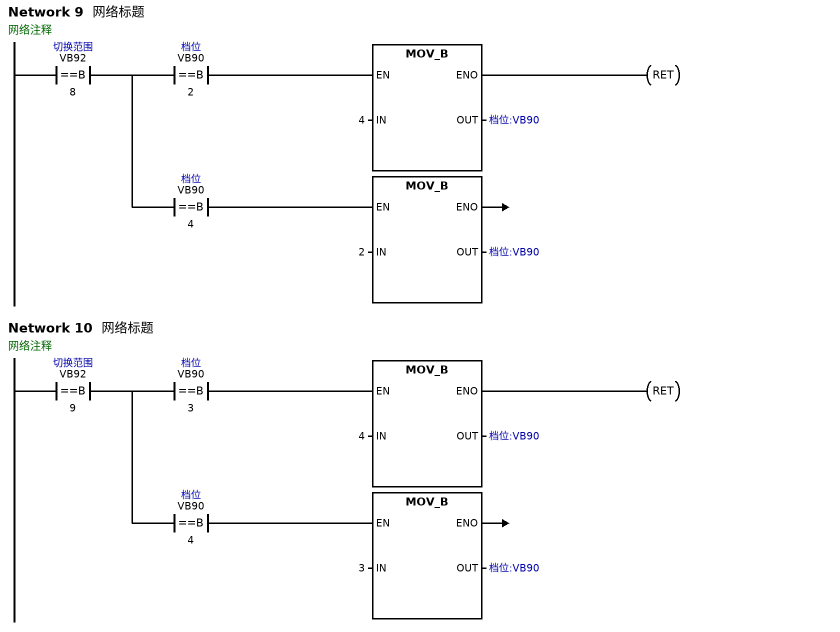
[picture p72: SBR19 networks 9-10]
Network 9 // 网络标题
// 网络注释
LDB=   切换范围:VB92, 8
LPS
AB=    档位:VB90, 2
MOVB   4, 档位:VB90
AENO
CRET
LPP
AB=    档位:VB90, 4
MOVB   2, 档位:VB90
Network 10 // 网络标题
// 网络注释
LDB=   切换范围:VB92, 9
LPS
AB=    档位:VB90, 3
MOVB   4, 档位:VB90
AENO
CRET
LPP
AB=    档位:VB90, 4
MOVB   3, 档位:VB90
END_SUBROUTINE_BLOCK

// SBR21: protected block, not included

SUBROUTINE_BLOCK ReCal:SBR22
TITLE=子程序注释
VAR_INPUT
Uo:REAL;	// LD0 
C‘:REAL;	// LD4 
K:REAL;	// LD8 
b:REAL;	// LD12 
END_VAR
VAR_OUTPUT
U‘:REAL;	// LD16 
A’:REAL;	// LD20 
END_VAR
VAR
mid:REAL;	// LD24 
END_VAR
BEGIN
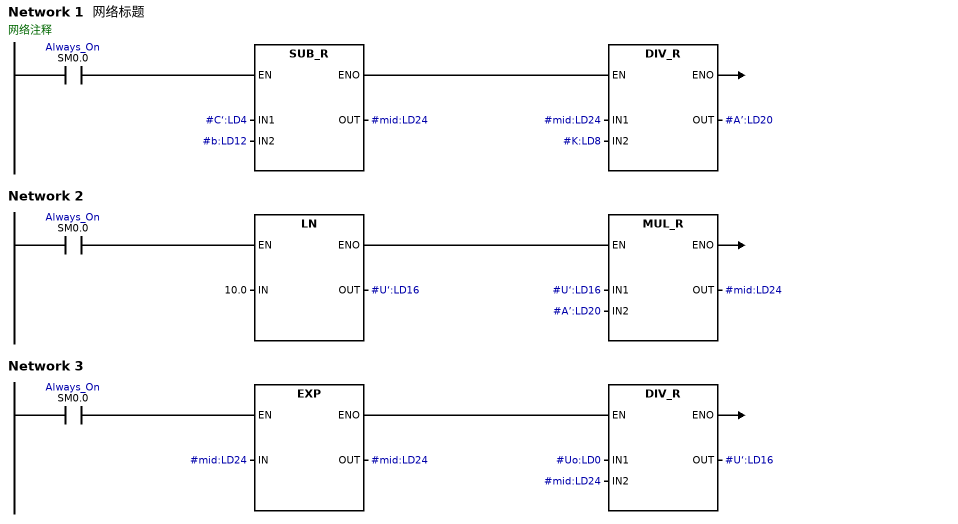
Network 1 // 网络标题
// 网络注释
LD     Always_On:SM0.0
MOVR   #C‘:LD4, #mid:LD24
AENO
-R     #b:LD12, #mid:LD24
AENO
MOVR   #mid:LD24, #A’:LD20
/R     #K:LD8, #A’:LD20
Network 2
LD     Always_On:SM0.0
LN     10.0, #U‘:LD16
AENO
MOVR   #U‘:LD16, #mid:LD24
*R     #A’:LD20, #mid:LD24
Network 3
LD     Always_On:SM0.0
EXP    #mid:LD24, #mid:LD24
AENO
MOVR   #Uo:LD0, #U‘:LD16
/R     #mid:LD24, #U‘:LD16
Network 4 // 网络标题
// 网络注释
END_SUBROUTINE_BLOCK

SUBROUTINE_BLOCK 标准R_I:SBR23
TITLE=子程序注释
VAR_INPUT
R_H:REAL;	// LD0 
R_L:REAL;	// LD4 
I_H:WORD;	// LW8 
I_L:WORD;	// LW10 
Input:REAL;	// LD12 
END_VAR
VAR_OUTPUT
output:WORD;	// LW16 
END_VAR
BEGIN
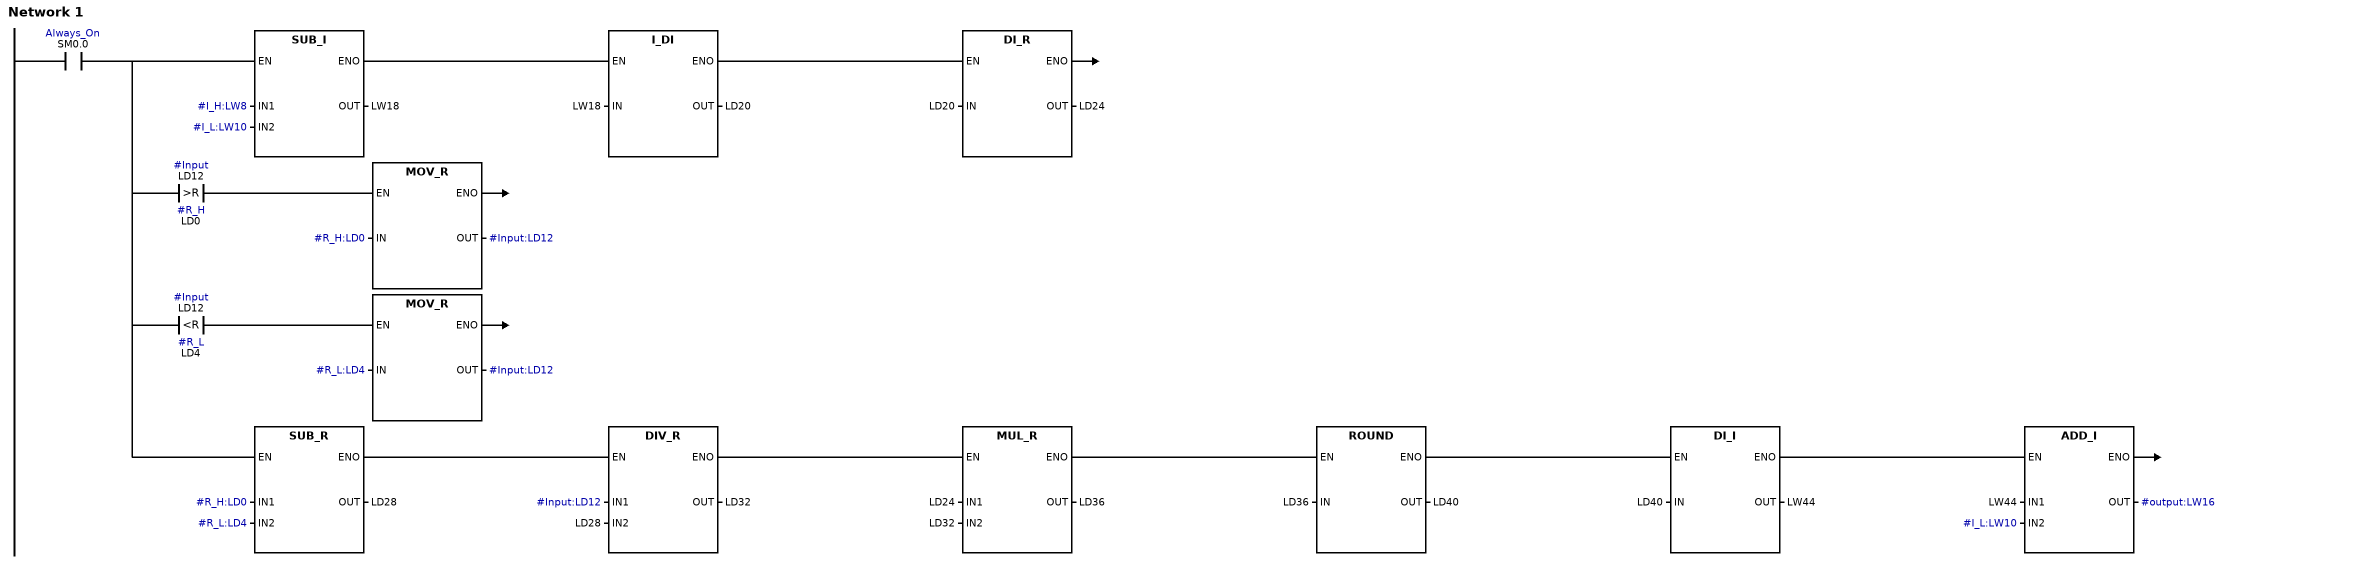
Network 1
LD     Always_On:SM0.0
LPS
MOVW   #I_H:LW8, LW18
AENO
-I     #I_L:LW10, LW18
AENO
ITD    LW18, LD20
AENO
DTR    LD20, LD24
LRD
AR>    #Input:LD12, #R_H:LD0
MOVR   #R_H:LD0, #Input:LD12
LRD
AR<    #Input:LD12, #R_L:LD4
MOVR   #R_L:LD4, #Input:LD12
LPP
MOVR   #R_H:LD0, LD28
AENO
-R     #R_L:LD4, LD28
AENO
MOVR   #Input:LD12, LD32
AENO
/R     LD28, LD32
AENO
MOVR   LD24, LD36
AENO
*R     LD32, LD36
AENO
ROUND  LD36, LD40
AENO
DTI    LD40, LW44
AENO
MOVW   LW44, #output:LW16
+I     #I_L:LW10, #output:LW16
END_SUBROUTINE_BLOCK

SUBROUTINE_BLOCK 动态管控参数:SBR24
TITLE=子程序注释
BEGIN
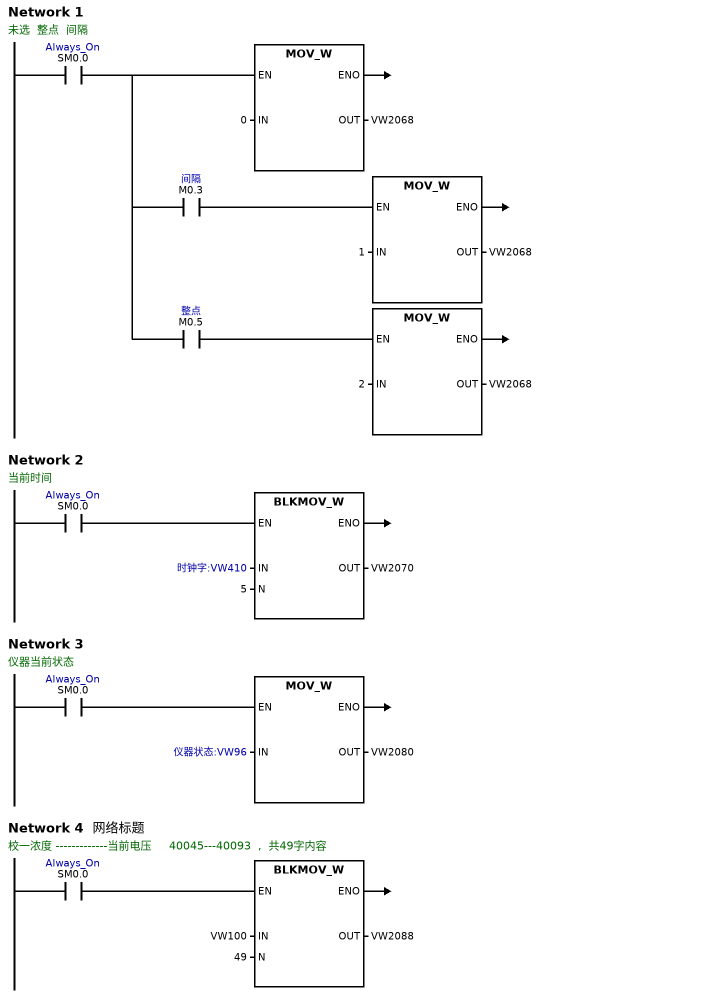
Network 1
//  未选  整点  间隔
LD     Always_On:SM0.0
LPS
MOVW   0, VW2068
A      间隔:M0.3
MOVW   1, VW2068
LPP
A      整点:M0.5
MOVW   2, VW2068
Network 2
// 当前时间
LD     Always_On:SM0.0
BMW    时钟字:VW410, VW2070, 5
Network 3
// 仪器当前状态
LD     Always_On:SM0.0
MOVW   仪器状态:VW96, VW2080
Network 4 // 网络标题
// 校一浓度 -------------当前电压     40045---40093  ,  共49字内容
LD     Always_On:SM0.0
BMW    VW100, VW2088, 49
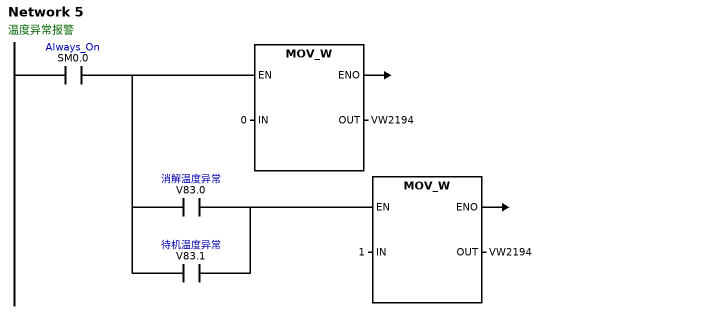
Network 5
// 温度异常报警
LD     Always_On:SM0.0
MOVW   0, VW2194
LD     消解温度异常:V83.0
O      待机温度异常:V83.1
ALD
MOVW   1, VW2194
Network 6
// 电极电压异常报警
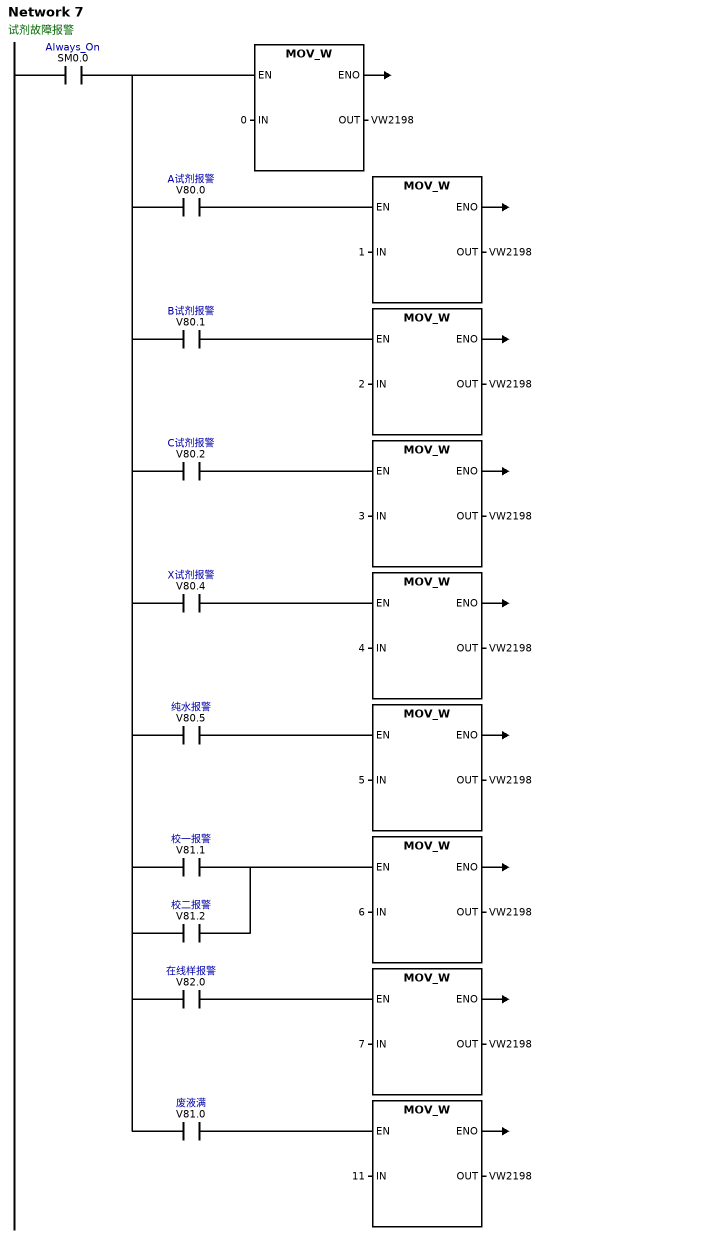
Network 7
// 试剂故障报警
LD     Always_On:SM0.0
LPS
MOVW   0, VW2198
A      A试剂报警:V80.0
MOVW   1, VW2198
LRD
A      B试剂报警:V80.1
MOVW   2, VW2198
LRD
A      C试剂报警:V80.2
MOVW   3, VW2198
LRD
A      X试剂报警:V80.4
MOVW   4, VW2198
LRD
A      纯水报警:V80.5
MOVW   5, VW2198
LRD
LD     校一报警:V81.1
O      校二报警:V81.2
ALD
MOVW   6, VW2198
LPP
LPS
A      在线样报警:V82.0
MOVW   7, VW2198
LPP
A      废液满:V81.0
MOVW   11, VW2198
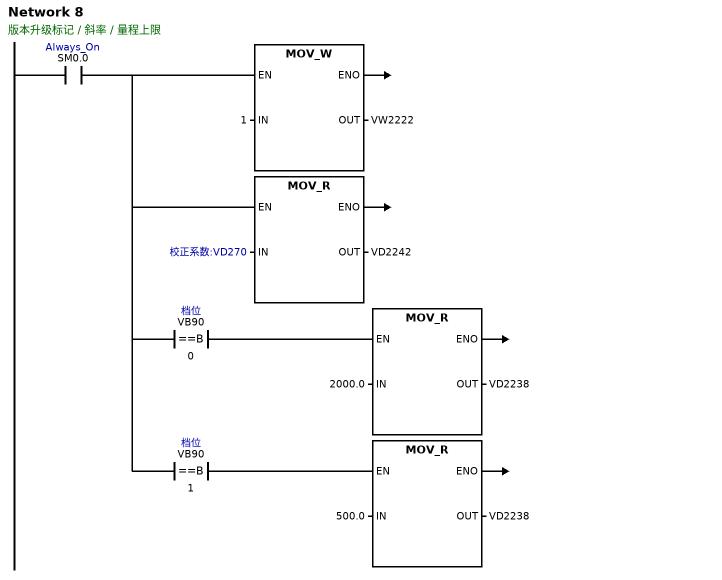
Network 8
// 版本升级标记
// 斜率
// 量程上限
LD     Always_On:SM0.0
LPS
MOVW   1, VW2222
MOVR   校正系数:VD270, VD2242
AB=    档位:VB90, 0
MOVR   2000.0, VD2238
LPP
AB=    档位:VB90, 1
MOVR   500.0, VD2238
END_SUBROUTINE_BLOCK

SUBROUTINE_BLOCK 设备状态:SBR25
TITLE=子程序注释
BEGIN
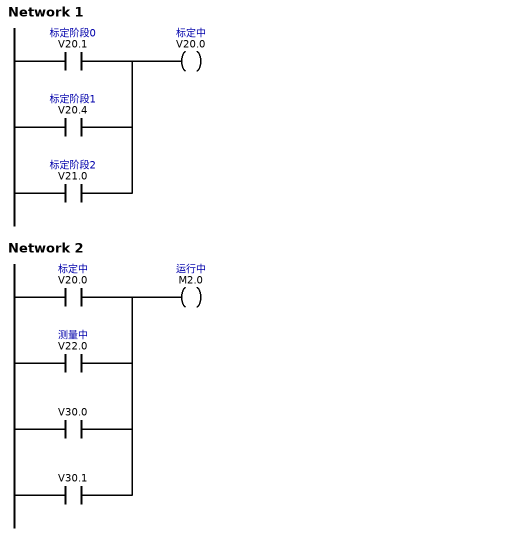
Network 1
LD     标定阶段0:V20.1
O      标定阶段1:V20.4
O      标定阶段2:V21.0
=      标定中:V20.0
Network 2
LD     标定中:V20.0
O      测量中:V22.0
O      V30.0
O      V30.1
=      运行中:M2.0
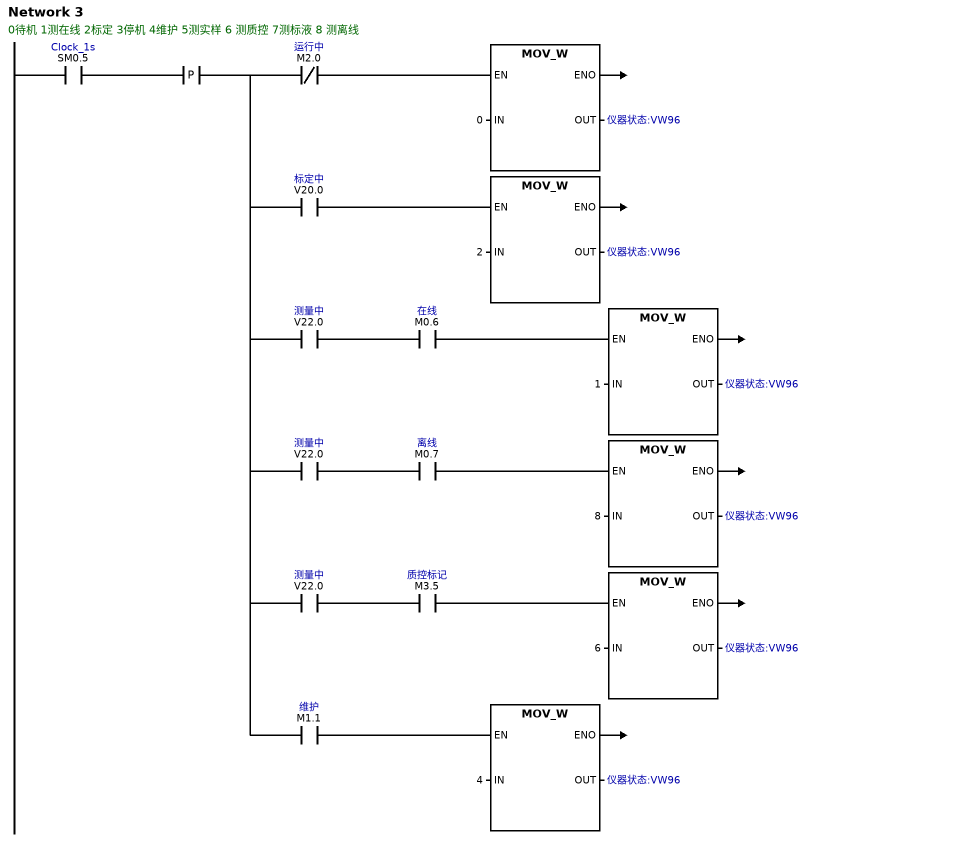
Network 3
// 0待机 1测在线 2标定 3停机 4维护 5测实样 6 测质控 7测标液 8 测离线
LD     Clock_1s:SM0.5
EU
LPS
AN     运行中:M2.0
MOVW   0, 仪器状态:VW96
LRD
A      标定中:V20.0
MOVW   2, 仪器状态:VW96
LRD
A      测量中:V22.0
A      在线:M0.6
MOVW   1, 仪器状态:VW96
LRD
A      测量中:V22.0
A      离线:M0.7
MOVW   8, 仪器状态:VW96
LRD
A      测量中:V22.0
A      质控标记:M3.5
MOVW   6, 仪器状态:VW96
LPP
A      维护:M1.1
MOVW   4, 仪器状态:VW96
END_SUBROUTINE_BLOCK

SUBROUTINE_BLOCK 密码:SBR26
TITLE=子程序注释
BEGIN
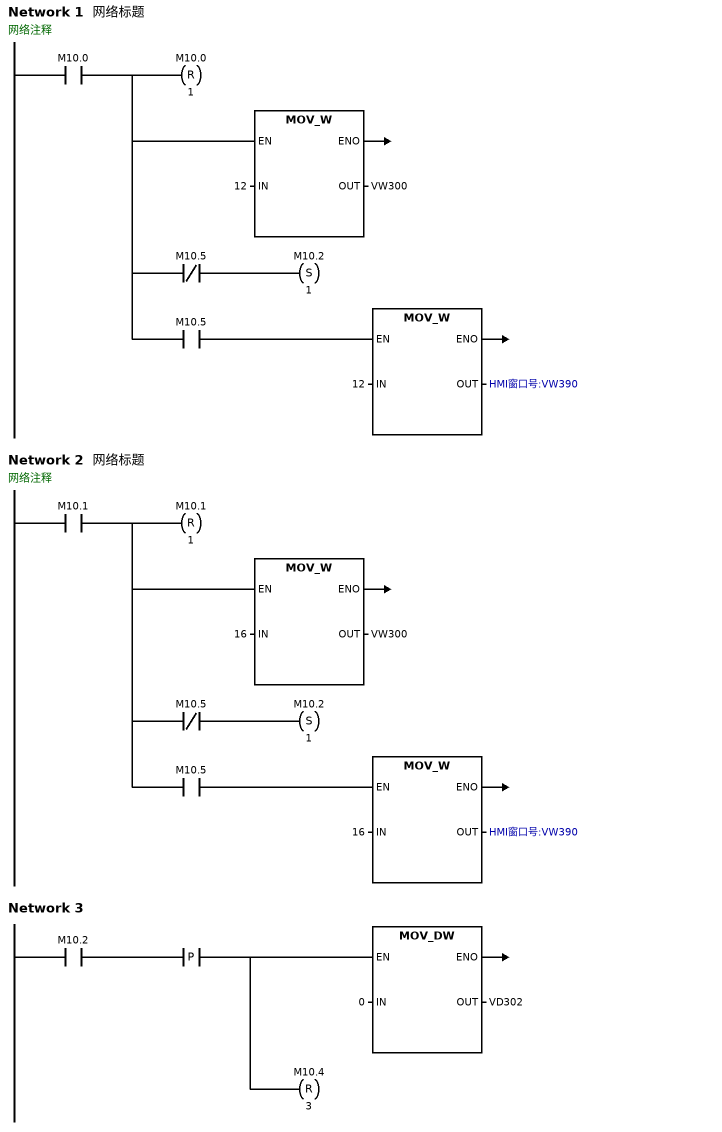
Network 1 // 网络标题
// 网络注释
LD     M10.0
LPS
R      M10.0, 1
MOVW   12, VW300
AN     M10.5
S      M10.2, 1
LPP
A      M10.5
MOVW   12, HMI窗口号:VW390
Network 2 // 网络标题
// 网络注释
LD     M10.1
LPS
R      M10.1, 1
MOVW   16, VW300
AN     M10.5
S      M10.2, 1
LPP
A      M10.5
MOVW   16, HMI窗口号:VW390
Network 3
LD     M10.2
EU
MOVD   0, VD302
R      M10.4, 3
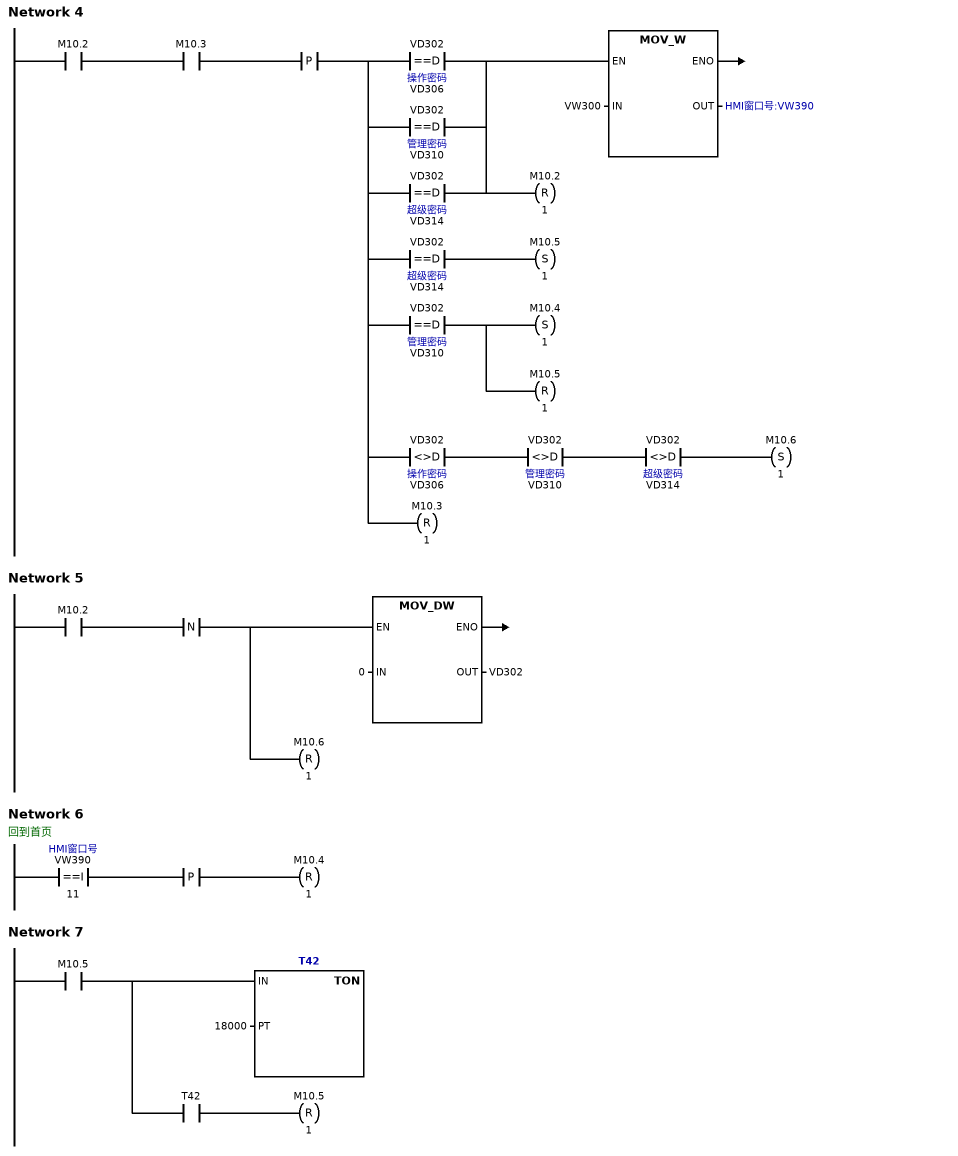
Network 4
LD     M10.2
A      M10.3
EU
LPS
LDD=   VD302, 操作密码:VD306
OD=    VD302, 管理密码:VD310
OD=    VD302, 超级密码:VD314
ALD
MOVW   VW300, HMI窗口号:VW390
R      M10.2, 1
LRD
AD=    VD302, 超级密码:VD314
S      M10.5, 1
LRD
AD=    VD302, 管理密码:VD310
S      M10.4, 1
R      M10.5, 1
LPP
LPS
AD<>   VD302, 操作密码:VD306
AD<>   VD302, 管理密码:VD310
AD<>   VD302, 超级密码:VD314
S      M10.6, 1
LPP
R      M10.3, 1
Network 5
LD     M10.2
ED
MOVD   0, VD302
R      M10.6, 1
Network 6
// 回到首页
LDW=   HMI窗口号:VW390, 11
EU
R      M10.4, 1
Network 7
LD     M10.5
TON    T42, 18000
A      T42
R      M10.5, 1
END_SUBROUTINE_BLOCK

SUBROUTINE_BLOCK 单位转换:SBR27
TITLE=子程序注释
BEGIN
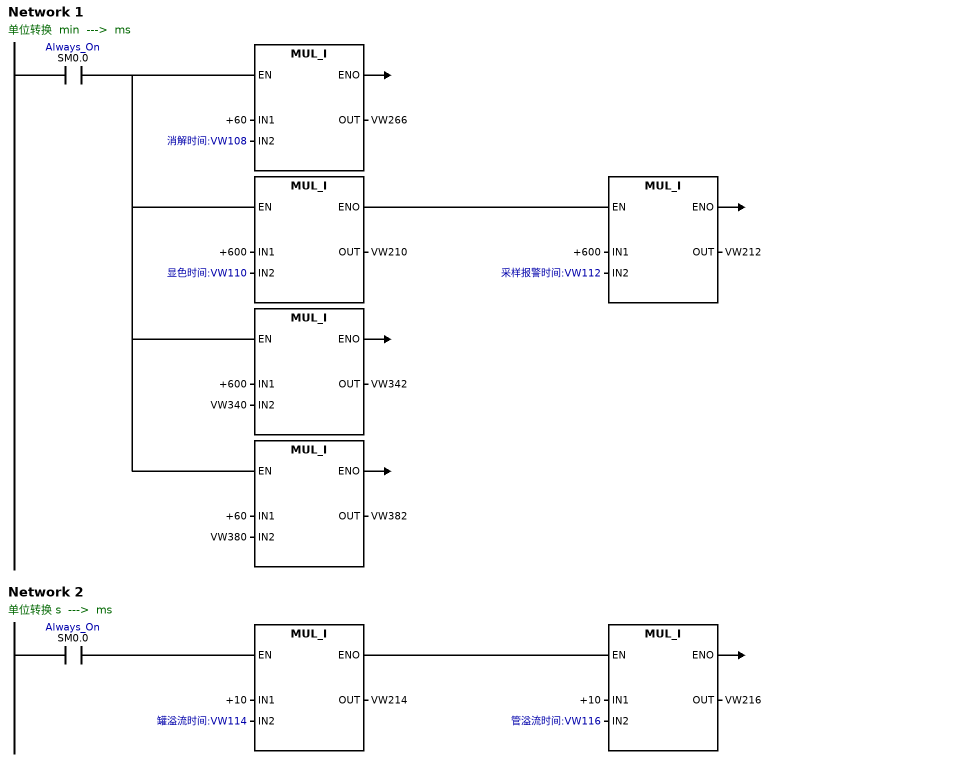
Network 1
// 单位转换  min  --->  ms
// (network saved uncompiled; LAD cells follow)
// row 0: c0 -| |- Always_On:SM0.0 v  c1 --  c2 [MUL_I EN:=power@row0, IN1:=+60, IN2:=消解时间:VW108, ENO=>power, OUT=>VW266]  c3 ->
// row 1: c0 ^v  c2 [box]
// row 2: c0 ^v  c1 --  c2 [MUL_I EN:=power@row2, IN1:=+600, IN2:=显色时间:VW110, ENO=>power, OUT=>VW210]  c3 --  c4 --  c5 [MUL_I EN:=power@row2, IN1:=+600, IN2:=采样报警时间:VW112, ENO=>power, OUT=>VW212]  c6 ->
// row 3: c0 ^v  c2 [box]  c5 [box]
// row 4: c0 ^v  c1 --  c2 [MUL_I EN:=power@row4, IN1:=+600, IN2:=VW340, ENO=>power, OUT=>VW342]  c3 ->
// row 5: c0 ^v  c2 [box]
// row 6: c0 ^  c1 --  c2 [MUL_I EN:=power@row6, IN1:=+60, IN2:=VW380, ENO=>power, OUT=>VW382]  c3 ->
// row 7: c2 [box]
Network 2
// 单位转换 s  --->  ms
LD     Always_On:SM0.0
MOVW   +10, VW214
AENO
*I     罐溢流时间:VW114, VW214
AENO
MOVW   +10, VW216
*I     管溢流时间:VW116, VW216
Network 3 // 网络标题
// 网络注释
END_SUBROUTINE_BLOCK

SUBROUTINE_BLOCK 读时钟:SBR28
TITLE=
BEGIN
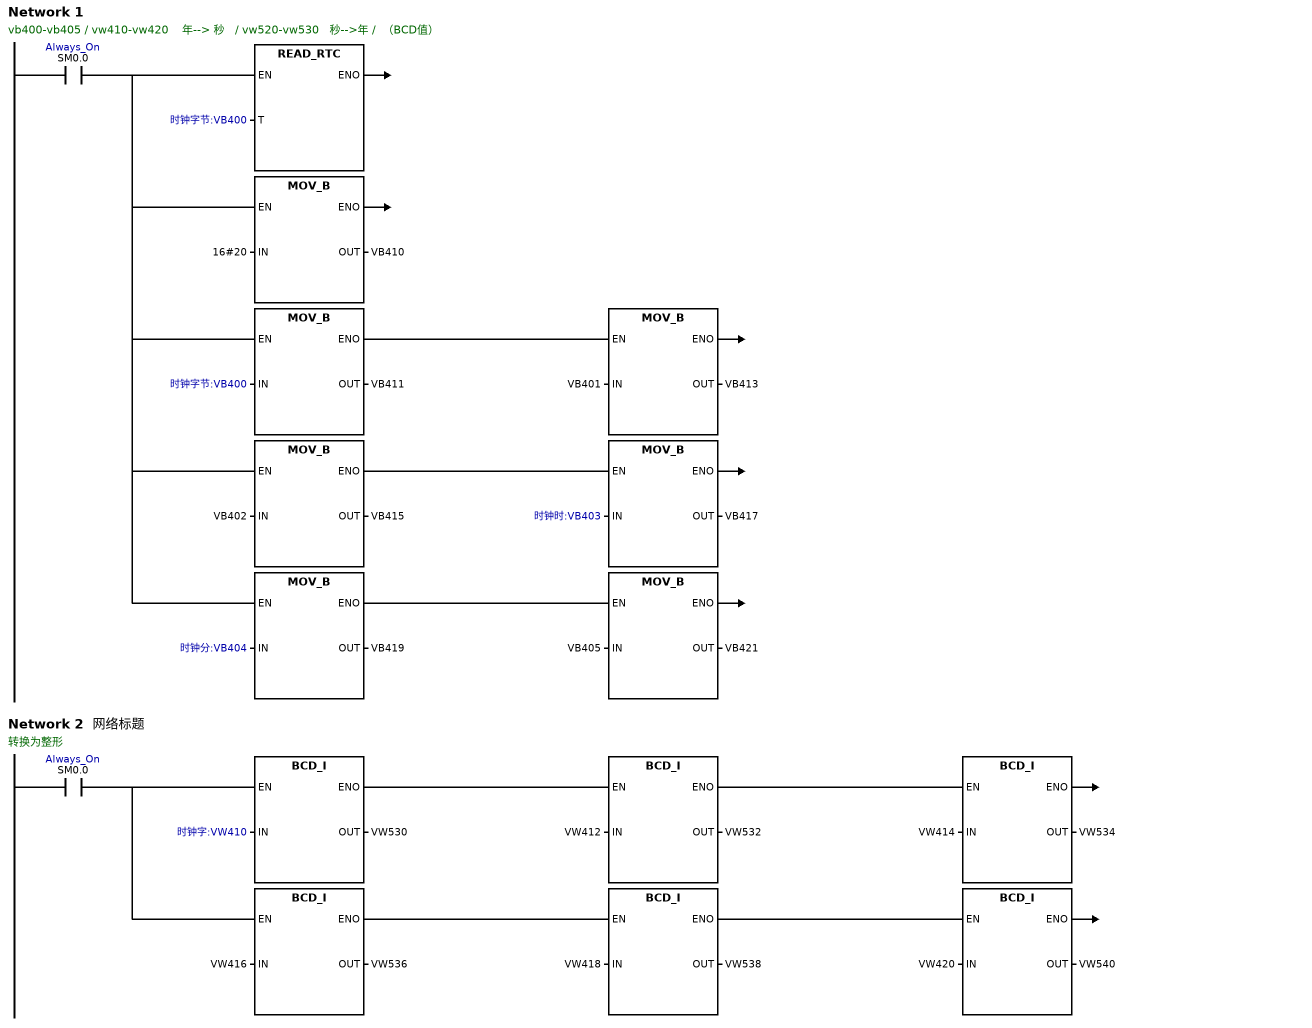
Network 1
// vb400-vb405
// vw410-vw420    年--> 秒  
// vw520-vw530   秒-->年
//  （BCD值）
LD     Always_On:SM0.0
LPS
TODR   时钟字节:VB400
MOVB   16#20, VB410
MOVB   时钟字节:VB400, VB411
AENO
MOVB   VB401, VB413
LRD
MOVB   VB402, VB415
AENO
MOVB   时钟时:VB403, VB417
LPP
MOVB   时钟分:VB404, VB419
AENO
MOVB   VB405, VB421
Network 2 // 网络标题
// 转换为整形
LD     Always_On:SM0.0
LPS
MOVW   时钟字:VW410, VW530
AENO
BCDI   VW530
AENO
MOVW   VW412, VW532
AENO
BCDI   VW532
AENO
MOVW   VW414, VW534
BCDI   VW534
LPP
MOVW   VW416, VW536
AENO
BCDI   VW536
AENO
MOVW   VW418, VW538
AENO
BCDI   VW538
AENO
MOVW   VW420, VW540
BCDI   VW540
END_SUBROUTINE_BLOCK

SUBROUTINE_BLOCK M7抽推比色皿:SBR29
TITLE=
VAR_INPUT
抽:BOOL;	// L0.0 
时间:WORD;	// LW1 
END_VAR
VAR_IN_OUT
启动位:BOOL;	// L3.0 
END_VAR
VAR_OUTPUT
结束位:BOOL;	// L3.1 
END_VAR
BEGIN
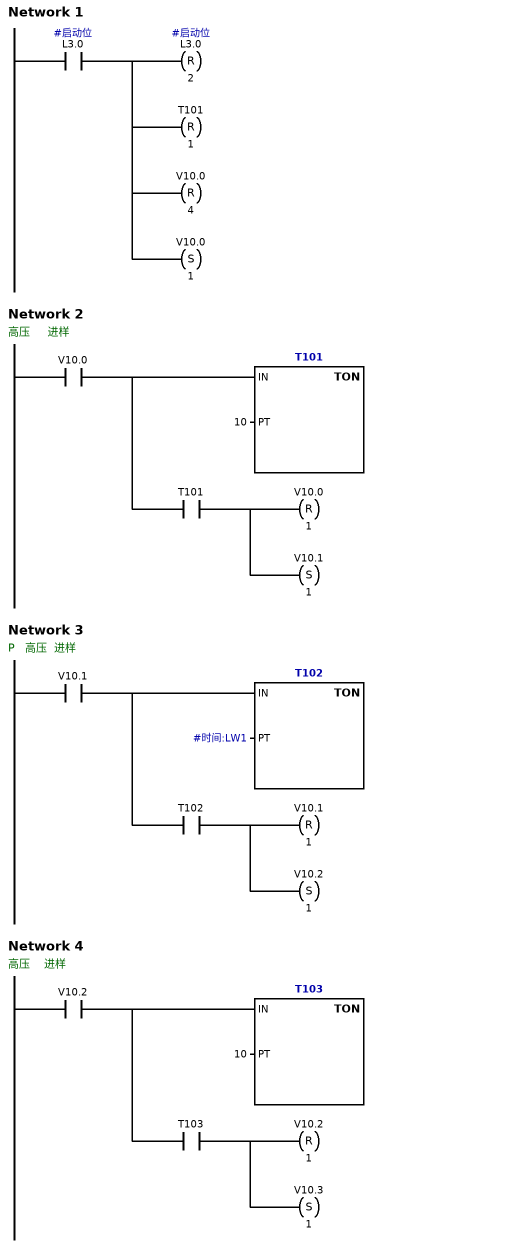
Network 1
LD     #启动位:L3.0
R      #启动位:L3.0, 2
R      T101, 1
R      V10.0, 4
S      V10.0, 1
Network 2
// 高压     进样
LD     V10.0
TON    T101, 10
A      T101
R      V10.0, 1
S      V10.1, 1
Network 3
// P   高压  进样
LD     V10.1
TON    T102, #时间:LW1
A      T102
R      V10.1, 1
S      V10.2, 1
Network 4
// 高压    进样
LD     V10.2
TON    T103, 10
A      T103
R      V10.2, 1
S      V10.3, 1
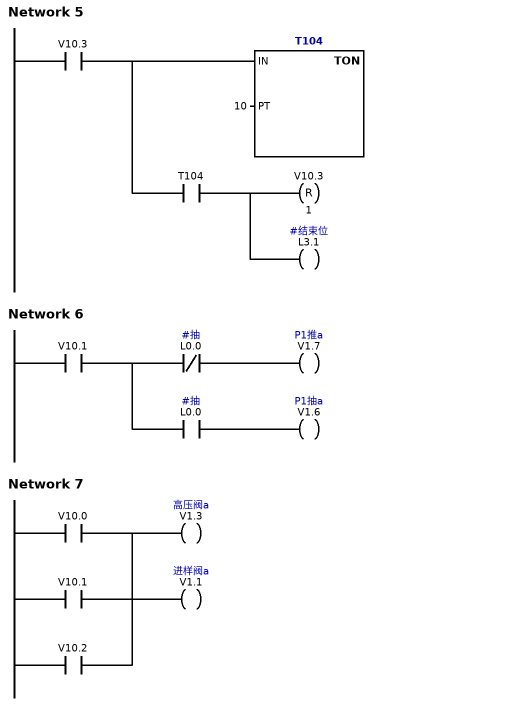
Network 5
LD     V10.3
TON    T104, 10
A      T104
R      V10.3, 1
=      #结束位:L3.1
Network 6
LD     V10.1
LPS
AN     #抽:L0.0
=      P1推a:V1.7
LPP
A      #抽:L0.0
=      P1抽a:V1.6
Network 7
LD     V10.0
O      V10.1
O      V10.2
=      高压阀a:V1.3
=      进样阀a:V1.1
Network 8 // 网络标题
// 网络注释
END_SUBROUTINE_BLOCK

// SBR30: protected block, not included

// SBR31: protected block, not included

// SBR32: protected block, not included

SUBROUTINE_BLOCK M8抽推多联体:SBR33
TITLE=
VAR_INPUT
抽:BOOL;	// L0.0 
时间:WORD;	// LW1 
END_VAR
VAR_IN_OUT
启动位:BOOL;	// L3.0 
END_VAR
VAR_OUTPUT
结束位:BOOL;	// L3.1 
阀:BOOL;	// L3.2 
END_VAR
BEGIN
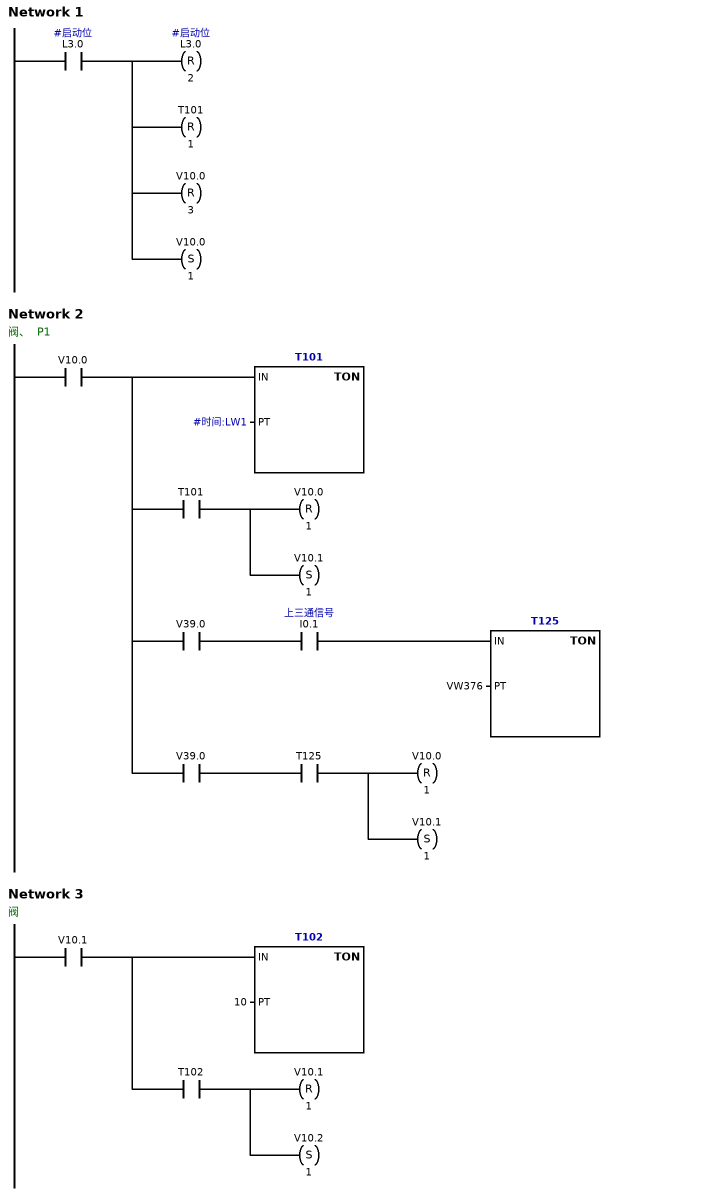
Network 1
LD     #启动位:L3.0
R      #启动位:L3.0, 2
R      T101, 1
R      V10.0, 3
S      V10.0, 1
Network 2
// 阀、  P1
LD     V10.0
LPS
TON    T101, #时间:LW1
A      T101
R      V10.0, 1
S      V10.1, 1
LRD
A      V39.0
A      上三通信号:I0.1
TON    T125, VW376
LPP
A      V39.0
A      T125
R      V10.0, 1
S      V10.1, 1
Network 3
// 阀
LD     V10.1
TON    T102, 10
A      T102
R      V10.1, 1
S      V10.2, 1
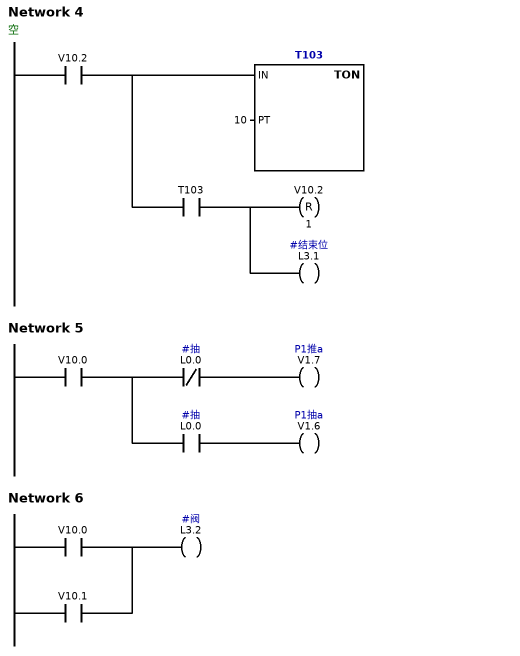
Network 4
// 空
LD     V10.2
TON    T103, 10
A      T103
R      V10.2, 1
=      #结束位:L3.1
Network 5
LD     V10.0
LPS
AN     #抽:L0.0
=      P1推a:V1.7
LPP
A      #抽:L0.0
=      P1抽a:V1.6
Network 6
LD     V10.0
O      V10.1
=      #阀:L3.2
Network 7 // 网络标题
// 网络注释
END_SUBROUTINE_BLOCK

SUBROUTINE_BLOCK 复位:SBR34
TITLE=级别越高复位内容越多
VAR_INPUT
level:BYTE;	// LB0 
END_VAR
BEGIN
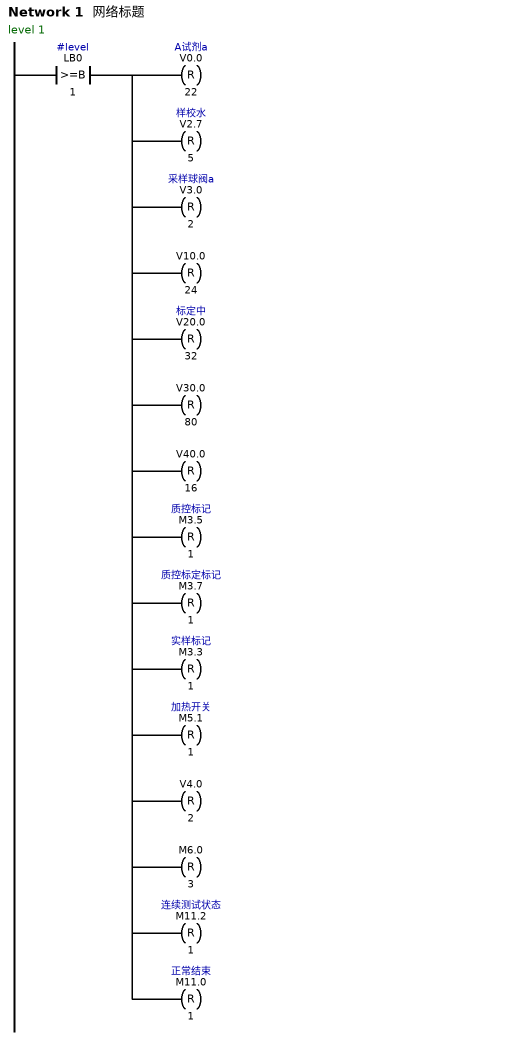
Network 1 // 网络标题
// level 1
LDB>=  #level:LB0, 1
R      A试剂a:V0.0, 22
R      样校水:V2.7, 5
R      采样球阀a:V3.0, 2
R      V10.0, 24
R      标定中:V20.0, 32
R      V30.0, 80
R      V40.0, 16
R      质控标记:M3.5, 1
R      质控标定标记:M3.7, 1
R      实样标记:M3.3, 1
R      加热开关:M5.1, 1
R      V4.0, 2
R      M6.0, 3
R      连续测试状态:M11.2, 1
R      正常结束:M11.0, 1
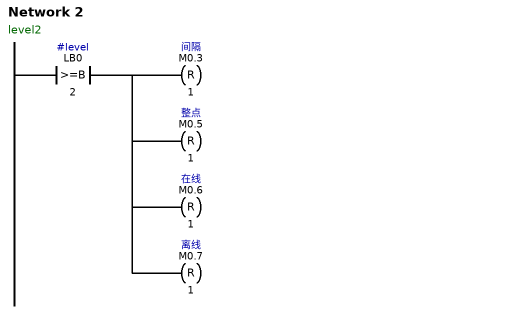
Network 2
// level2
LDB>=  #level:LB0, 2
R      间隔:M0.3, 1
R      整点:M0.5, 1
R      在线:M0.6, 1
R      离线:M0.7, 1
END_SUBROUTINE_BLOCK

SUBROUTINE_BLOCK 流程步骤名:SBR35
TITLE=子程序注释
BEGIN
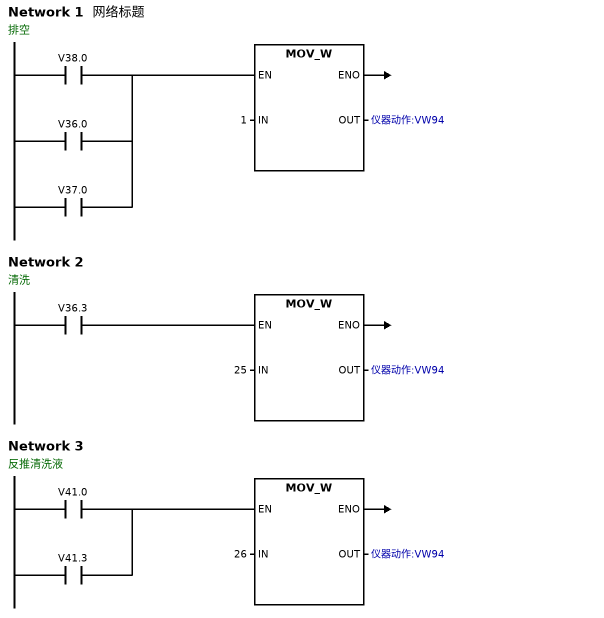
Network 1 // 网络标题
// 排空
LD     V38.0
O      V36.0
O      V37.0
MOVW   1, 仪器动作:VW94
Network 2
// 清洗
LD     V36.3
MOVW   25, 仪器动作:VW94
Network 3
// 反推清洗液
LD     V41.0
O      V41.3
MOVW   26, 仪器动作:VW94
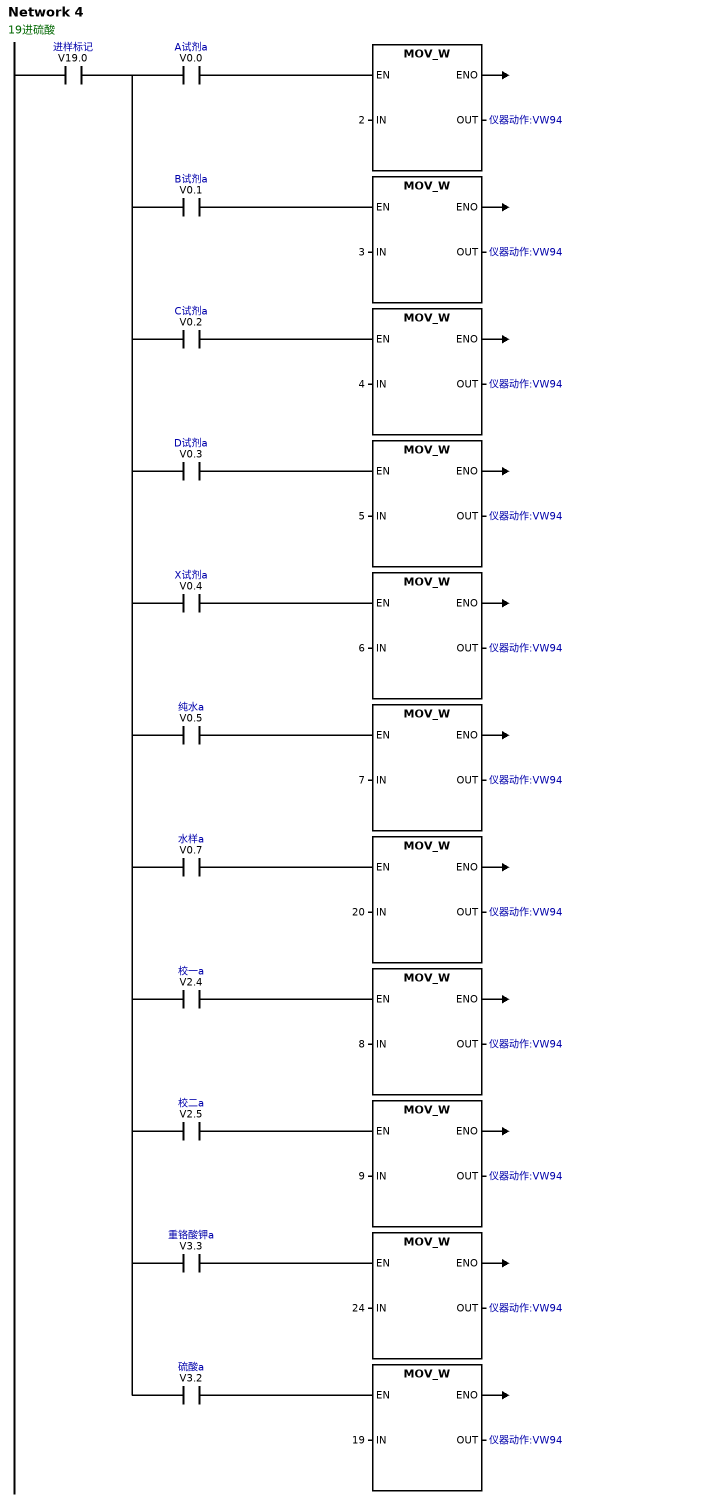
Network 4
// 19进硫酸
LD     进样标记:V19.0
LPS
A      A试剂a:V0.0
MOVW   2, 仪器动作:VW94
LRD
A      B试剂a:V0.1
MOVW   3, 仪器动作:VW94
LRD
A      C试剂a:V0.2
MOVW   4, 仪器动作:VW94
LRD
A      D试剂a:V0.3
MOVW   5, 仪器动作:VW94
LRD
A      X试剂a:V0.4
MOVW   6, 仪器动作:VW94
LRD
A      纯水a:V0.5
MOVW   7, 仪器动作:VW94
LRD
A      水样a:V0.7
MOVW   20, 仪器动作:VW94
LRD
A      校一a:V2.4
MOVW   8, 仪器动作:VW94
LRD
A      校二a:V2.5
MOVW   9, 仪器动作:VW94
LRD
A      重铬酸钾a:V3.3
MOVW   24, 仪器动作:VW94
LPP
A      硫酸a:V3.2
MOVW   19, 仪器动作:VW94
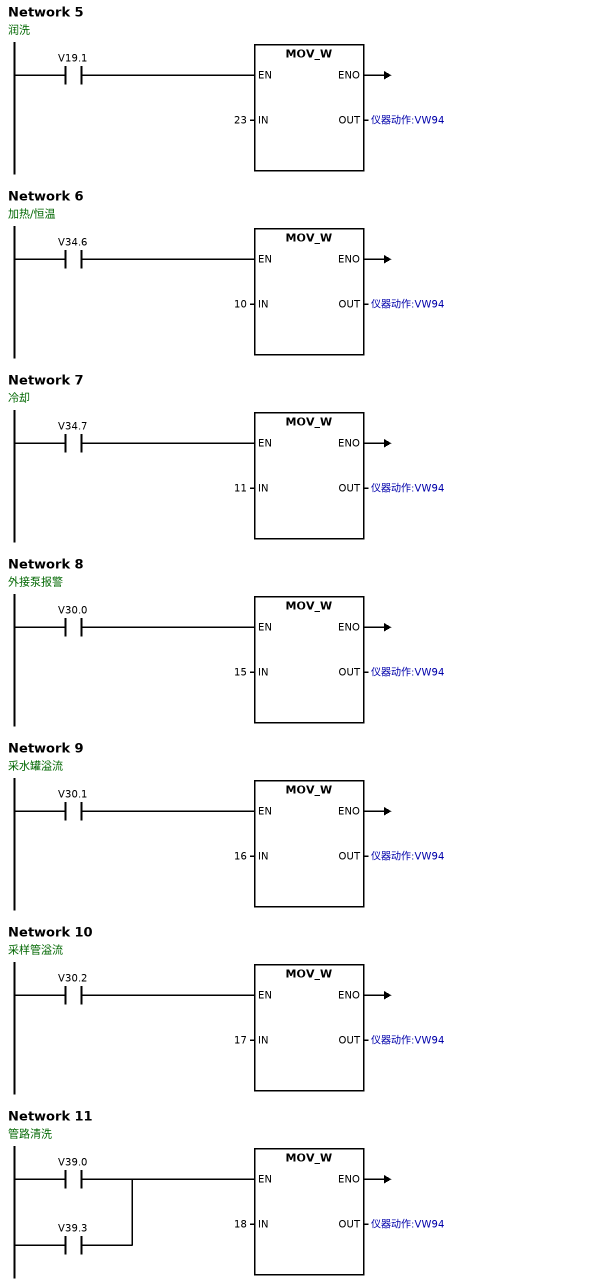
Network 5
// 润洗
LD     V19.1
MOVW   23, 仪器动作:VW94
Network 6
// 加热/恒温
LD     V34.6
MOVW   10, 仪器动作:VW94
Network 7
// 冷却
LD     V34.7
MOVW   11, 仪器动作:VW94
Network 8
// 外接泵报警
LD     V30.0
MOVW   15, 仪器动作:VW94
Network 9
// 采水罐溢流
LD     V30.1
MOVW   16, 仪器动作:VW94
Network 10
// 采样管溢流
LD     V30.2
MOVW   17, 仪器动作:VW94
Network 11
// 管路清洗
LD     V39.0
O      V39.3
MOVW   18, 仪器动作:VW94
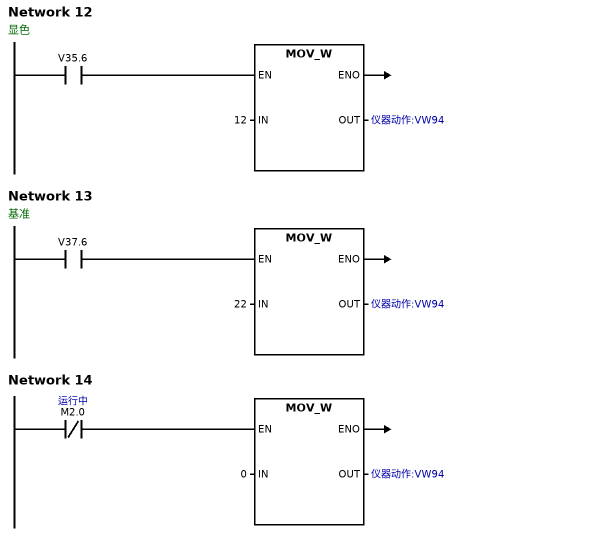
Network 12
// 显色
LD     V35.6
MOVW   12, 仪器动作:VW94
Network 13
// 基准
LD     V37.6
MOVW   22, 仪器动作:VW94
Network 14
LDN    运行中:M2.0
MOVW   0, 仪器动作:VW94
END_SUBROUTINE_BLOCK

SUBROUTINE_BLOCK 三层:SBR36
TITLE=子程序注释
BEGIN
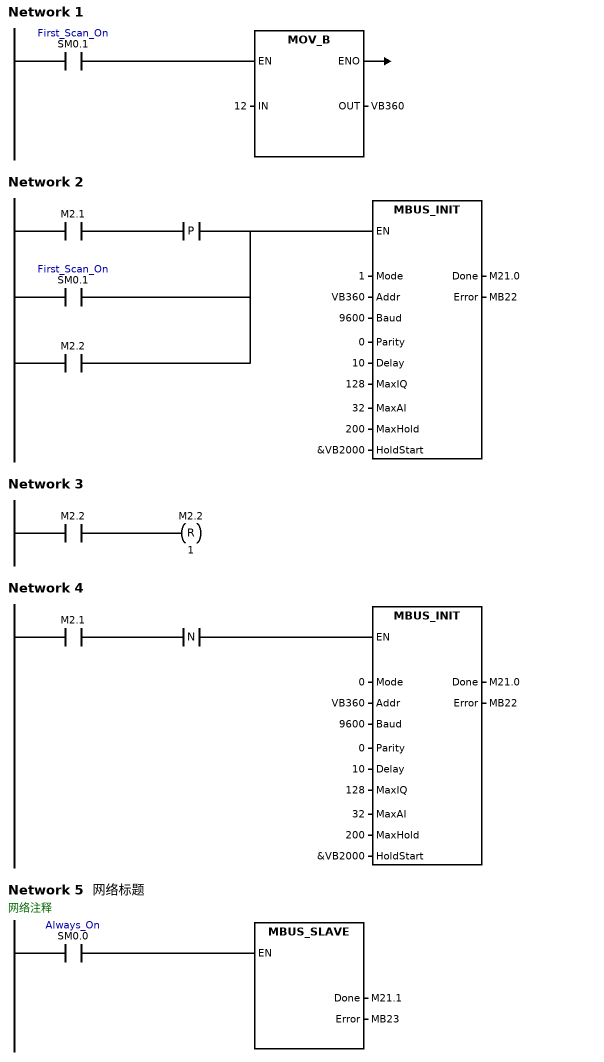
Network 1
LD     First_Scan_On:SM0.1
MOVB   12, VB360
Network 2
LD     M2.1
EU
O      First_Scan_On:SM0.1
O      M2.2
CALL   MBUS_INIT:SBR30, 1, VB360, 9600, 0, 10, 128, 32, 200, &VB2000, M21.0, MB22
Network 3
LD     M2.2
R      M2.2, 1
Network 4
LD     M2.1
ED
CALL   MBUS_INIT:SBR30, 0, VB360, 9600, 0, 10, 128, 32, 200, &VB2000, M21.0, MB22
Network 5 // 网络标题
// 网络注释
LD     Always_On:SM0.0
CALL   MBUS_SLAVE:SBR31, M21.1, MB23
END_SUBROUTINE_BLOCK

SUBROUTINE_BLOCK 计算A:SBR37
TITLE=
VAR_INPUT
显色1:REAL;	// LD0 
基准1:REAL;	// LD4 
END_VAR
VAR_OUTPUT
A1:REAL;	// LD8 
END_VAR
BEGIN
